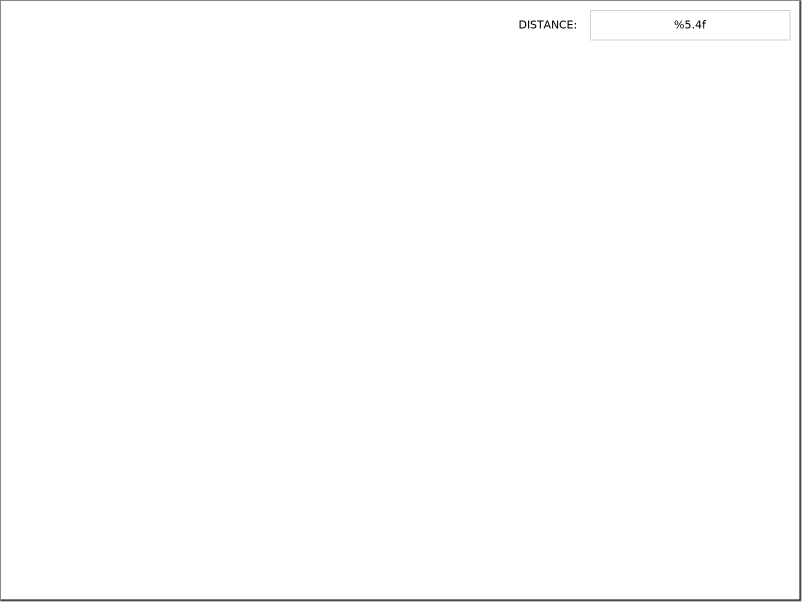
VISUALIZATION F29_Move_Relative  // 802x602
    Rectangle (0,0 800x600)
    Textfield (590,10 200x30), "%5.4f", text variable: MAIN.axes[MAIN.hmiAxisSelect].DISTANCE
        OnMouseClick: write MAIN.axes[MAIN.hmiAxisSelect].DISTANCE via Default
    Label (410,10 170x30), "DISTANCE:"
END_VISUALIZATION

(* stored: Version 1.1.0.1, ProductVersion 3.1.4022.7
   Visu F29_Move_Relative: Id {8a994c57-6cfc-42b5-981b-01533fb8df62} *)
